TYPE ST_AxisConfig :
STRUCT
	
	///////Axis Parameters//////
	fOverride			:	LREAL := 100;	//Controller override %
	fVelocity			:	LREAL;			//Velocity must be specified, no default used
	fAcceleration		:	LREAL;			//Not all FBs use, need to change this, 0 is NC default
	fDeceleration		:	LREAL;
	fPosition			:	LREAL;			//Used for absolute positioning	
	nHomeSeq			:	UINT;			//Homing sequence to perform

END_STRUCT
END_TYPE

(* stored: Version 1.1.0.1, ProductVersion 3.1.4022.12
   DUT ST_AxisConfig: Id {e00fe310-8ff8-452a-800a-823efa83b1a3} *)
